{attribute 'qualified_only'}
{attribute 'strict'}
{attribute 'to_string'}
TYPE E_TestEnum :
(
	Idle := 0,
	Starting,
	Running,
	Stopping,
	Pausing,
	Paused,
	Error,
	ErrorResetting
) UINT;
END_TYPE

(* stored: Version 1.1.0.1
   DUT E_TestEnum: Id {e8bbe942-eadb-4bfb-9fec-311a2dd23c3f} *)
